{attribute 'GeneratedUsingTerminal: KL2702'}
{attribute addProperty BoxType "KL2702"}
{attribute addProperty Id "Channel_1AT %Q*Channel_460B8C400Channel_2AT %Q*Channel_460B8C400"}
{attribute addProperty CRC "3701954066"}
{attribute addProperty Size "0"}
TYPE KL2702_DCA75612 :
STRUCT
	{attribute addProperty Name "Channel_1"}
	Channel_1 : Channel_460B8C40;
	{attribute addProperty Name "Channel_2"}
	Channel_2 : Channel_460B8C40;
END_STRUCT
END_TYPE

(* stored: Version 1.2.0.0, ProductVersion 3.1.4024.9
   DUT KL2702_DCA75612: Id {5272211d-9a4c-4c75-a478-ab09a6555740} *)
